FUNCTION_BLOCK FB_Encoder
VAR_INPUT
END_VAR
VAR_OUTPUT
END_VAR
VAR
END_VAR

END_FUNCTION_BLOCK

(* stored: Version 1.1.0.1
   POU FB_Encoder: Id {78e5da71-5f6e-4401-978d-f3722c3321b2}, SpecialFunc None *)
